// Swaps values of to variables
FUNCTION SwapByAddr : E_GeneralStatus
VAR_INPUT
	A : POINTER TO BYTE;
	B : POINTER TO BYTE;
	Length : DINT;
END_VAR
VAR
	Temp : POINTER TO BYTE;
END_VAR


IF A = 0 OR B = 0 THEN
	
	SwapByAddr := E_GeneralStatus.INPUT_ERROR;
	RETURN;
END_IF

Temp := __NEW(BYTE, Length);

MEMCPY(Temp, A, Length);
MEMCPY(A, B, Length);
MEMCPY(B, Temp, Length);

__DELETE(Temp);

SwapByAddr := E_GeneralStatus.DONE;

END_FUNCTION

(* stored: Version 1.1.0.1, ProductVersion 3.1.4024.11
   POU SwapByAddr: Id {8f7e6b3f-cfc8-4cf3-a66c-26ce49090c04}, SpecialFunc None *)
